FUNCTION_BLOCK FB_EL7047_Tuner
VAR_INPUT
    _stAxis             : REFERENCE TO ST_AxisStruct; 
    stTuningInputs      : ST_Tuning;
    
    // Intelligent Auto-Tune Parameters
    bExecuteAutoTune    : BOOL;
    bStepMode           : BOOL; // If TRUE, pauses after each pass
    bNextStep           : BOOL; // Trigger to proceed to the next pass
    nKpStartOverride    : UINT := 150;    // If > 0, overrides the L calculation (Beckhoff default is 150)
    nMaxCurrent_mA      : UINT := 0;      // 0x8010:01. If 0, the block reads the existing CoE value natively
    
    // Resonance Testing Velocity Range
    fTestVelocity       : LREAL := 7.5;   // Velocity where resonance occurs
    fTestDistance       : LREAL := 50.0;  // Distance to travel for measuring
    
    // Tuning Constraints
    fTnMin              : REAL := 0.3;    // ms
    fTnMax              : REAL := 1.0;    // ms
    nKiStart            : UINT := 1;
    nKiEnd              : UINT := 20;
    nKiStep             : UINT := 1;
    fKpReductionPct     : LREAL := 10.0;  // Reduce Kp by 10% per major loop
    nMaxKpIterations    : UINT := 5;      // How many times to reduce Kp
    
    // Manual Mode (Python ADS Server)
    bExecuteSingleTest  : BOOL; // Python triggers this to run just one pass and fill the array
    
    // Manual Parameter Application (HMI Staging Area)
    bApplyParams        : BOOL; // Trigger to write Staging Area to the drive
    nApplyMaxCurrent    : UINT; // The Current to write (auto-filled with CurrentRun after tuning)
    nApplyKp            : UINT; // The Kp to write (auto-filled with BestKp after tuning)
    nApplyKi            : UINT; // The Ki to write (auto-filled with BestKi after tuning)
    
    // Baseline Snapshot (HMI)
    bSaveBaseline       : BOOL; // Trigger to lock the current Best into the Baseline arrays
    bLoadBaseline       : BOOL; // Trigger to copy Baseline values into the Staging Area
    
    // Error Handling
    bContinueAfterError : BOOL; // Retry the failed step from the HMI
    bAbortTuning        : BOOL; // Abort tuning and return to Idle
END_VAR
VAR_OUTPUT
    bBusy               : BOOL;
    bDone               : BOOL;
    bError              : BOOL;
    nErrorId            : UDINT;
    
    // Run Results (Current Sweep)
    nCurrentRunMaxCurrent: UINT; // Shows what current was actually used for this test
    nBestKp             : UINT;
    nBestKi             : UINT;
    fBestResonanceScore : LREAL;
    
    nWorstKp            : UINT;
    nWorstKi            : UINT;
    fWorstResonanceScore: LREAL;
    
    // Baseline Snapshot (Manually saved)
    nBaselineMaxCurrent : UINT;
    nBaselineKp         : UINT;
    nBaselineKi         : UINT;
    fBaselineScore      : LREAL;
END_VAR
VAR
    // The high-speed 1ms buffer for ADS extraction or internal analysis
    aLoadData           : ARRAY[1..1000] OF INT; // InfoData 1 (Current Run)
    aBestLoadData       : ARRAY[1..1000] OF INT; // InfoData 1 (Best Run Snapshot)
    aWorstLoadData      : ARRAY[1..1000] OF INT; // InfoData 1 (Worst Run Snapshot)
    aBaselineLoadData   : ARRAY[1..1000] OF INT; // InfoData 1 (Locked Baseline Snapshot)
    
    aPowerData          : ARRAY[1..1000] OF INT; // InfoData 2
    nSampleCount        : UINT;
    
    // Internal State Machine and Motion Blocks
    eState              : E_TunerState;
    eNextState          : E_TunerState;
    eErrorSource        : E_TunerState; // Stores where the error occurred for retrying
    fbCoEWrite          : FB_EcCoESdoWrite;
    fbCoERead           : FB_EcCoESdoRead;
    fbMoveRelative      : MC_MoveRelative;
    fbSettleTimer       : TON;
    fbReadStatus        : MC_ReadStatus;
    
    // Loop trackers and internal calculations
    fMotorInductance    : LREAL; // Fetched natively from CoE
    nCurrentKp          : UINT;
    nCurrentKi          : UINT;
    nIteration          : UINT;
    fCurrentTn          : REAL;
    
    // CoE buffer
    nCoEWriteBuffer     : UINT;
    nTnCoEBuffer        : UINT;
    nCoEInductanceBuf   : UINT;
    
    // Math evaluation
    i                   : UINT;
    nMaxLoad            : INT; // Kept for visual reference if needed
    nMinLoad            : INT;
    fCurrentResonance   : LREAL; // Will now store Variance instead of Peak-to-Peak
    
    nStartIndex         : UINT;
    nEndIndex           : UINT;
    nWindowSize         : UINT;
    fSum                : LREAL;
    fMean               : LREAL;
    fVarianceSum        : LREAL;
    fDiff               : LREAL;
END_VAR

// Initialize FB parameters
fbCoEWrite(sNetId := _stAxis.stConfig.stCoEParameters.sEthCATNetId, nSlaveAddr := _stAxis.stConfig.stCoEParameters.nSlaveAdressDrive);
fbCoERead(sNetId := _stAxis.stConfig.stCoEParameters.sEthCATNetId, nSlaveAddr := _stAxis.stConfig.stCoEParameters.nSlaveAdressDrive);
fbMoveRelative(Axis := _stAxis.Axis, Velocity := fTestVelocity);
fbReadStatus(Axis := _stAxis.Axis, Enable := TRUE);

// Manual Baseline Trigger
IF bSaveBaseline THEN
    bSaveBaseline := FALSE;
    nBaselineMaxCurrent := nCurrentRunMaxCurrent;
    nBaselineKp := nBestKp;
    nBaselineKi := nBestKi;
    fBaselineScore := fBestResonanceScore;
    MEMCPY(ADR(aBaselineLoadData), ADR(aBestLoadData), SIZEOF(aBestLoadData));
END_IF

// Load Baseline to Staging Area
IF bLoadBaseline THEN
    bLoadBaseline := FALSE;
    nApplyMaxCurrent := nBaselineMaxCurrent;
    nApplyKp := nBaselineKp;
    nApplyKi := nBaselineKi;
END_IF

CASE eState OF
    E_TunerState.eIdle:
        IF bExecuteAutoTune THEN
            bBusy := TRUE;
            bDone := FALSE;
            bError := FALSE;
            nErrorId := 0;
            nIteration := 0;
            fBestResonanceScore := 999999999.0; // Initialize high for current run (Variance can be large)
            fWorstResonanceScore := 0.0;     // Initialize low for current run
            
            IF nKpStartOverride = 0 THEN
                eState := E_TunerState.eReadInductance;
            ELSE
                IF nMaxCurrent_mA = 0 THEN
                    eState := E_TunerState.eReadMaxCurrent;
                ELSE
                    nCurrentRunMaxCurrent := nMaxCurrent_mA;
                    eState := E_TunerState.eWriteMaxCurrent;
                END_IF
            END_IF
            
        ELSIF bExecuteSingleTest THEN
            // Manual single-shot mode (for Python plotting)
            bBusy := TRUE;
            bDone := FALSE;
            bError := FALSE;
            nSampleCount := 0;
            MEMSET(ADR(aLoadData), 0, SIZEOF(aLoadData));
            MEMSET(ADR(aPowerData), 0, SIZEOF(aPowerData));
            
            fbMoveRelative.Distance := fTestDistance;
            fbMoveRelative.Execute := TRUE;
            eState := E_TunerState.eMoveFwd;
            
        ELSIF bApplyParams THEN
            // HMI Manual Application of Params
            bBusy := TRUE;
            bDone := FALSE;
            bError := FALSE;
            eState := E_TunerState.eApplyManualCurrent;
        END_IF
        
    E_TunerState.eReadInductance:
        fbCoERead.nIndex := 16#8010;
        fbCoERead.nSubIndex := 16#0A; // Assumed Inductance sub-index (Check EL7047 Manual)
        fbCoERead.pDstBuf := ADR(nCoEInductanceBuf);
        fbCoERead.cbBufLen := SIZEOF(nCoEInductanceBuf);
        fbCoERead.bExecute := TRUE;
        
        IF NOT fbCoERead.bBusy AND NOT fbCoERead.bError THEN
            fbCoERead.bExecute := FALSE;
            // Assumes value is in 0.01 mH resolution. Convert to Henry.
            fMotorInductance := UINT_TO_LREAL(nCoEInductanceBuf) * 0.00001; 
            
            IF nMaxCurrent_mA = 0 THEN
                eState := E_TunerState.eReadMaxCurrent;
            ELSE
                nCurrentRunMaxCurrent := nMaxCurrent_mA;
                eState := E_TunerState.eWriteMaxCurrent;
            END_IF
            
        ELSIF fbCoERead.bError THEN
            eErrorSource := eState;
            nErrorId := fbCoERead.nErrId;
            eState := E_TunerState.eError;
        END_IF
        
    E_TunerState.eReadMaxCurrent:
        fbCoERead.nIndex := 16#8010;
        fbCoERead.nSubIndex := 16#01; 
        fbCoERead.pDstBuf := ADR(nCurrentRunMaxCurrent);
        fbCoERead.cbBufLen := SIZEOF(nCurrentRunMaxCurrent);
        fbCoERead.bExecute := TRUE;
        
        IF NOT fbCoERead.bBusy AND NOT fbCoERead.bError THEN
            fbCoERead.bExecute := FALSE;
            IF nKpStartOverride = 0 THEN
                eState := E_TunerState.eCalcStartKp;
            ELSE
                nCurrentKi := nKiStart;
                eState := E_TunerState.eWriteKp;
            END_IF
        ELSIF fbCoERead.bError THEN
            eErrorSource := eState;
            nErrorId := fbCoERead.nErrId;
            eState := E_TunerState.eError;
        END_IF
        
    E_TunerState.eWriteMaxCurrent:
        fbCoEWrite.nIndex := 16#8010;
        fbCoEWrite.nSubIndex := 16#01;
        nCoEWriteBuffer := nMaxCurrent_mA;
        fbCoEWrite.pSrcBuf := ADR(nCoEWriteBuffer);
        fbCoEWrite.cbBufLen := SIZEOF(nCoEWriteBuffer);
        fbCoEWrite.bExecute := TRUE;
        
        IF NOT fbCoEWrite.bBusy AND NOT fbCoEWrite.bError THEN
            fbCoEWrite.bExecute := FALSE;
            IF nKpStartOverride = 0 THEN
                eState := E_TunerState.eCalcStartKp;
            ELSE
                nCurrentKi := nKiStart;
                eState := E_TunerState.eWriteKp;
            END_IF
        ELSIF fbCoEWrite.bError THEN
            nErrorId := fbCoEWrite.nErrId;
            eErrorSource := eState;
            eState := E_TunerState.eError;
        END_IF
        
    E_TunerState.eCalcStartKp:
        // Kp = 10000 * 2pi * L
        nCurrentKp := LREAL_TO_UINT(10000.0 * 2.0 * 3.14159265359 * fMotorInductance);
        nCurrentKi := nKiStart;
        eState := E_TunerState.eWriteKp;
        
    E_TunerState.eWriteKp:
        fbCoEWrite.nIndex := 16#8011;
        fbCoEWrite.nSubIndex := 16#01;
        nCoEWriteBuffer := nCurrentKp;
        fbCoEWrite.pSrcBuf := ADR(nCoEWriteBuffer);
        fbCoEWrite.cbBufLen := SIZEOF(nCoEWriteBuffer);
        fbCoEWrite.bExecute := TRUE;
        
        IF NOT fbCoEWrite.bBusy AND NOT fbCoEWrite.bError THEN
            fbCoEWrite.bExecute := FALSE;
            eState := E_TunerState.eWriteKi;
        ELSIF fbCoEWrite.bError THEN
            nErrorId := fbCoEWrite.nErrId;
            eErrorSource := eState;
            eState := E_TunerState.eError;
        END_IF
        
    E_TunerState.eWriteKi:
        fbCoEWrite.nIndex := 16#8011;
        fbCoEWrite.nSubIndex := 16#02;
        nCoEWriteBuffer := nCurrentKi;
        fbCoEWrite.pSrcBuf := ADR(nCoEWriteBuffer);
        fbCoEWrite.cbBufLen := SIZEOF(nCoEWriteBuffer);
        fbCoEWrite.bExecute := TRUE;
        
        IF NOT fbCoEWrite.bBusy AND NOT fbCoEWrite.bError THEN
            fbCoEWrite.bExecute := FALSE;
            eState := E_TunerState.eReadTn;
        ELSIF fbCoEWrite.bError THEN
            nErrorId := fbCoEWrite.nErrId;
            eErrorSource := eState;
            eState := E_TunerState.eError;
        END_IF
        
    E_TunerState.eReadTn:
        fbCoERead.nIndex := 16#9010;
        fbCoERead.nSubIndex := 16#0E;
        fbCoERead.pDstBuf := ADR(nTnCoEBuffer);
        fbCoERead.cbBufLen := SIZEOF(nTnCoEBuffer);
        fbCoERead.bExecute := TRUE;
        
        IF NOT fbCoERead.bBusy AND NOT fbCoERead.bError THEN
            fbCoERead.bExecute := FALSE;
            fCurrentTn := UINT_TO_REAL(nTnCoEBuffer) * 0.01;
            eState := E_TunerState.eEvaluateTn;
        ELSIF fbCoERead.bError THEN
            nErrorId := fbCoERead.nErrId;
            eErrorSource := eState;
            eState := E_TunerState.eError;
        END_IF
        
    E_TunerState.eEvaluateTn:
        // Enforce Beckhoff bounds (0.3 to 1.0 ms)
        IF fCurrentTn >= fTnMin AND fCurrentTn <= fTnMax THEN
            nSampleCount := 0;
            MEMSET(ADR(aLoadData), 0, SIZEOF(aLoadData));
            MEMSET(ADR(aPowerData), 0, SIZEOF(aPowerData));
            
            fbMoveRelative.Distance := fTestDistance;
            fbMoveRelative.Execute := TRUE;
            eState := E_TunerState.eMoveFwd;
        ELSE
            // Skip this Ki since Tn is out of bounds
            eState := E_TunerState.eEvaluateResonance; 
        END_IF
        
    E_TunerState.eMoveFwd:
        // Stall Protection
        IF stTuningInputs.bStall THEN
            fbMoveRelative.Execute := FALSE;
            _stAxis.stControl.bStop := TRUE; // Let FB_Axis safely halt the motor
            nErrorId := 16#7047; // Custom Stall ErrorID
            eErrorSource := eState;
            eState := E_TunerState.eError;
        END_IF
        
        // Record high-speed arrays only during pure constant velocity
        IF fbReadStatus.ConstantVelocity THEN
            IF nSampleCount < 1000 THEN
                nSampleCount := nSampleCount + 1;
                aLoadData[nSampleCount] := stTuningInputs.nInfoData1;
                aPowerData[nSampleCount] := stTuningInputs.nInfoData2;
            END_IF
        END_IF
        
        IF fbMoveRelative.Done THEN
            fbMoveRelative.Execute := FALSE;
            eState := E_TunerState.eWaitMoveFwd;
        ELSIF fbMoveRelative.Error THEN
            nErrorId := fbMoveRelative.ErrorID;
            eErrorSource := eState;
            eState := E_TunerState.eError;
        END_IF
        
    E_TunerState.eWaitMoveFwd:
        // Delay before returning
        fbSettleTimer(IN := TRUE, PT := T#500MS);
        IF fbSettleTimer.Q THEN
            fbSettleTimer(IN := FALSE);
            fbMoveRelative.Distance := -fTestDistance;
            fbMoveRelative.Execute := TRUE;
            eState := E_TunerState.eMoveBwd;
        END_IF
        
    E_TunerState.eMoveBwd:
        // Stall Protection
        IF stTuningInputs.bStall THEN
            fbMoveRelative.Execute := FALSE;
            _stAxis.stControl.bStop := TRUE; // Let FB_Axis safely halt the motor
            nErrorId := 16#7047; // Custom Stall ErrorID
            eErrorSource := eState;
            eState := E_TunerState.eError;
        END_IF
        
        // Record high-speed arrays only during pure constant velocity
        IF fbReadStatus.ConstantVelocity THEN
            IF nSampleCount < 1000 THEN
                nSampleCount := nSampleCount + 1;
                aLoadData[nSampleCount] := stTuningInputs.nInfoData1;
                aPowerData[nSampleCount] := stTuningInputs.nInfoData2;
            END_IF
        END_IF
        
        IF fbMoveRelative.Done THEN
            fbMoveRelative.Execute := FALSE;
            IF bExecuteSingleTest THEN
                bBusy := FALSE;
                bDone := TRUE;
                eState := E_TunerState.eIdle;
            ELSE
                eState := E_TunerState.eEvaluateResonance;
            END_IF
        ELSIF fbMoveRelative.Error THEN
            nErrorId := fbMoveRelative.ErrorID;
            eErrorSource := eState;
            eState := E_TunerState.eError;
        END_IF
        
    E_TunerState.eEvaluateResonance:
        // Calculate Variance of the Load Angle (Data is guaranteed to be purely Constant Velocity)
        fCurrentResonance := 0.0;
        IF nSampleCount > 1 THEN
            // 1. Calculate the Mean
            fSum := 0.0;
            FOR i := 1 TO nSampleCount DO
                fSum := fSum + INT_TO_LREAL(aLoadData[i]);
            END_FOR
            fMean := fSum / UINT_TO_LREAL(nSampleCount);
            
            // 2. Calculate Variance (Sum of Squared Differences)
            fVarianceSum := 0.0;
            FOR i := 1 TO nSampleCount DO
                fDiff := INT_TO_LREAL(aLoadData[i]) - fMean;
                fVarianceSum := fVarianceSum + (fDiff * fDiff);
            END_FOR
            
            // The score is the variance. Lower is mathematically smoother.
            fCurrentResonance := fVarianceSum / UINT_TO_LREAL(nSampleCount);
            
            // Save if it's the smoothest run yet
            IF fCurrentResonance < fBestResonanceScore THEN
                fBestResonanceScore := fCurrentResonance;
                nBestKp := nCurrentKp;
                nBestKi := nCurrentKi;
                MEMCPY(ADR(aBestLoadData), ADR(aLoadData), SIZEOF(aLoadData));
            END_IF
            
            // Save if it's the worst run
            IF fCurrentResonance > fWorstResonanceScore THEN
                fWorstResonanceScore := fCurrentResonance;
                nWorstKp := nCurrentKp;
                nWorstKi := nCurrentKi;
                MEMCPY(ADR(aWorstLoadData), ADR(aLoadData), SIZEOF(aLoadData));
            END_IF
        END_IF
        
        // Loop iteration logic
        nCurrentKi := nCurrentKi + nKiStep;
        IF nCurrentKi <= nKiEnd THEN
            eNextState := E_TunerState.eWriteKi;
        ELSE
            nIteration := nIteration + 1;
            IF nIteration <= nMaxKpIterations THEN
                nCurrentKp := LREAL_TO_UINT(UINT_TO_LREAL(nCurrentKp) * (1.0 - (fKpReductionPct / 100.0)));
                nCurrentKi := nKiStart;
                eNextState := E_TunerState.eWriteKp;
            ELSE
                eNextState := E_TunerState.eApplyBestParams;
            END_IF
        END_IF
        
        IF bStepMode THEN
            eState := E_TunerState.eWaitNextStep;
        ELSE
            eState := eNextState;
        END_IF
        
    E_TunerState.eWaitNextStep:
        IF bNextStep THEN
            bNextStep := FALSE;
            eState := eNextState;
        ELSIF bAbortTuning THEN
            bAbortTuning := FALSE;
            eState := E_TunerState.eIdle;
        END_IF
        
    E_TunerState.eApplyBestParams:
        // Optimization complete. 
        // We populate the manual apply inputs with the winner, so the user can review and click apply.
        nApplyKp := nBestKp;
        nApplyKi := nBestKi;
        nApplyMaxCurrent := nCurrentRunMaxCurrent;
        bBusy := FALSE;
        bDone := TRUE;
        eState := E_TunerState.eIdle;
        
    E_TunerState.eApplyManualCurrent:
        fbCoEWrite.nIndex := 16#8010;
        fbCoEWrite.nSubIndex := 16#01;
        nCoEWriteBuffer := nApplyMaxCurrent;
        fbCoEWrite.pSrcBuf := ADR(nCoEWriteBuffer);
        fbCoEWrite.cbBufLen := SIZEOF(nCoEWriteBuffer);
        fbCoEWrite.bExecute := TRUE;
        
        IF NOT fbCoEWrite.bBusy AND NOT fbCoEWrite.bError THEN
            fbCoEWrite.bExecute := FALSE;
            eState := E_TunerState.eApplyManualKp;
        ELSIF fbCoEWrite.bError THEN
            nErrorId := fbCoEWrite.nErrId;
            eErrorSource := eState;
            eState := E_TunerState.eError;
        END_IF
        
    E_TunerState.eApplyManualKp:
        fbCoEWrite.nIndex := 16#8011;
        fbCoEWrite.nSubIndex := 16#01;
        nCoEWriteBuffer := nApplyKp;
        fbCoEWrite.pSrcBuf := ADR(nCoEWriteBuffer);
        fbCoEWrite.cbBufLen := SIZEOF(nCoEWriteBuffer);
        fbCoEWrite.bExecute := TRUE;
        
        IF NOT fbCoEWrite.bBusy AND NOT fbCoEWrite.bError THEN
            fbCoEWrite.bExecute := FALSE;
            eState := E_TunerState.eApplyManualKi;
        ELSIF fbCoEWrite.bError THEN
            nErrorId := fbCoEWrite.nErrId;
            eErrorSource := eState;
            eState := E_TunerState.eError;
        END_IF
        
    E_TunerState.eApplyManualKi:
        fbCoEWrite.nIndex := 16#8011;
        fbCoEWrite.nSubIndex := 16#02;
        nCoEWriteBuffer := nApplyKi;
        fbCoEWrite.pSrcBuf := ADR(nCoEWriteBuffer);
        fbCoEWrite.cbBufLen := SIZEOF(nCoEWriteBuffer);
        fbCoEWrite.bExecute := TRUE;
        
        IF NOT fbCoEWrite.bBusy AND NOT fbCoEWrite.bError THEN
            fbCoEWrite.bExecute := FALSE;
            bApplyParams := FALSE; // Reset trigger
            bBusy := FALSE;
            bDone := TRUE;
            eState := E_TunerState.eIdle;
        ELSIF fbCoEWrite.bError THEN
            nErrorId := fbCoEWrite.nErrId;
            eErrorSource := eState;
            eState := E_TunerState.eError;
        END_IF
        
    E_TunerState.eError:
        bBusy := FALSE;
        bError := TRUE;
        fbCoERead.bExecute := FALSE;
        fbCoEWrite.bExecute := FALSE;
        fbMoveRelative.Execute := FALSE;
        
        IF bAbortTuning THEN
            bAbortTuning := FALSE;
            bError := FALSE;
            nErrorId := 0;
            eState := E_TunerState.eIdle;
        ELSIF bContinueAfterError THEN
            bContinueAfterError := FALSE;
            bError := FALSE;
            bBusy := TRUE;
            nErrorId := 0;
            eState := eErrorSource; // Retry the exact step that failed
        END_IF
END_CASE

END_FUNCTION_BLOCK

(* stored: Version 1.1.0.1
   POU FB_EL7047_Tuner: Id {2768c7ae-4a0c-4a4c-8b12-4d3efb5f2e6e}, SpecialFunc None *)
